FUNCTION_BLOCK F_XOR (* standard bitwise boolean function (xor) *)
  (* Standard: 61131-3; Classification: standard bitwise boolean function *)
  (* Version 1.0, 2009-09-14, 4DIAC-IDE, 4DIAC-Consortium *)
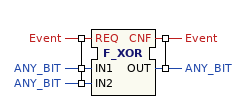
  EVENT_INPUT
    REQ WITH IN1, IN2; (* Service Request *)
  END_EVENT
  EVENT_OUTPUT
    CNF WITH OUT; (* Confirmation of Requested Service *)
  END_EVENT
  VAR_INPUT
    IN1 : ANY_BIT; (* Input *)
    IN2 : ANY_BIT; (* Input *)
  END_VAR
  VAR_OUTPUT
    OUT : ANY_BIT; (* Output *)
  END_VAR
  (* Service APPLICATION/RESOURCE: standard bitwise boolean function (xor) *)
END_FUNCTION_BLOCK
